(* CODESYS project NTC-Tester-Techmicron.project
   Version: 0.0.0.0
   Title: NTC-Tester-Techmicron
   Author: ekoru

Project tree, tasks and I/O mapping:
  MyController : TM241CE40R, Schneider Electric, order no. TM241CE40R, version 5.0.8.2
    application Application
      libraries: Network, 3.5.7.0 (3S - Smart Software Solutions GmbH)
      task MAST (cyclic, interval 20 ms, priority 15, watchdog 100 ms x 1) calls Input, Output, Auto_Sequence, Man_Sequence, DMM_Connection, Test_Result
      global variables GVL
      program Input [LD]
      program Output [LD]
      program Auto_Sequence [LD]
      program Man_Sequence [LD]
      program DMM_Connection [LD]
      program Test_Result [LD]
    DI : Digital Inputs, Schneider Electric, version 5.0.8.2
        input  idwDI_IDW0 : DWORD  // IDW0
        input  ibDI_IB1 : BYTE  // IB1
    DQ : Digital Outputs, Schneider Electric, version 5.0.8.2
        output qwDQ_QW0 : WORD  // QW0
        output qbDQ_QB1 : BYTE  // QB1
    Counters : Counters, Schneider Electric, version 5.0.8.2
    Pulse_Generators : Pulse Generators, Schneider Electric, version 5.0.8.2
    Cartridge_1 : Cartridge, Schneider Electric, version 5.0.8.2
    Cartridge_2 : Cartridge, Schneider Electric, version 5.0.8.2
    IO_Bus : IO bus - TM3, Schneider Electric, version 5.0.8.2
    COM_Bus : COM bus, Schneider Electric, version 5.0.8.2
    Ethernet_1 : Ethernet Network, Schneider Electric, version 5.0.8.2
        settings: IPAddress = [192, 168, 1, 10]; SubnetMask = [255, 255, 255, 0]; WebServer = TRUE; FTP Server = FALSE; SoMachine Protocol = TRUE; Modbus Server = FALSE; NetManage Protocol = TRUE; SNMP protocol = FALSE; Enable Routing = FALSE; WebVisu protocol = FALSE; DHCP Server Active = TRUE
    Serial_Line_1 : Serial line, Schneider Electric, version 5.0.8.2
      Machine_Expert_Network_Manager : Machine Expert-Network Manager, Schneider Electric, version 4.0.0.3
    Serial_Line_2 : Serial line, Schneider Electric, version 5.0.8.2
      Modbus_Manager : Modbus Manager, Schneider Electric, version 4.0.0.3
*)

// MyController/Application/GVL
{attribute 'qualified_only'}
VAR_GLOBAL
	// Input
	// S1
	Cyl_A_min AT %IX0.1: BOOL;
	// S2
	Cyl_A_max AT %IX0.0: BOOL;
	// S3
	Cyl_B_min AT %IX0.2: BOOL;
	// S4
	Cyl_B_max AT %IX0.3: BOOL;
	// S5
	Jig_Sensor AT %IX0.4: BOOL;
	// S6
	Sw_EMG AT %IX0.8: BOOL;
	// S7
	Sw_Auto AT %IX0.9: BOOL;
	// S8
	Sw_PB_Left AT %IX0.10: BOOL;
	// S9
	Sw_PB_Right AT %IX0.11: BOOL;
	// Timer Cyl A min
	Timer_Cyl_A_min: BOOL;
	Timer_Cyl_A_max: BOOL;
	Timer_Cyl_B_min: BOOL;
	Timer_Cyl_B_max: BOOL;
	Timer_Jig_Sensor: BOOL;
	Trigger_Cycle: BOOL;
	
	// Output
	Led_Red_1 AT %QX0.0: BOOL;
	Led_Red_2 AT %QX0.1: BOOL;
	Led_Red_3 AT %QX0.2: BOOL;
	Led_Red_4 AT %QX0.3: BOOL;
	Led_Green_1 AT %QX0.4: BOOL;
	Led_Green_2 AT %QX0.5: BOOL;
	Led_Green_3 AT %QX0.6: BOOL;
	Led_Green_4 AT %QX0.7: BOOL;
	Sol_Cyl_A AT %QX0.8: BOOL;
	Sol_Cyl_B AT %QX0.9: BOOL;
	Buzzer AT %QX0.10: BOOL;
	Coil_K1 AT %QX0.11: BOOL;
	Coil_K2 AT %QX0.12: BOOL;
	Coil_K3 AT %QX0.13: BOOL;
	Coil_K4 AT %QX0.14: BOOL;
	
	// Sequence
	Seq_Cyl_A_Forward: BOOL;
	Seq_Cyl_B_Down: BOOL;
	Seq_Test_1: BOOL;
	Seq_Test_2: BOOL;
	Seq_Test_3: BOOL;
	Seq_Test_4: BOOL;
	Seq_Cyl_B_Up: BOOL;
	Seq_Cyl_A_Backward: BOOL;
	Seq_Done: BOOL;
	Sw_PB_Right_Cycle: BOOL;
	Man_Done: BOOL;
	Man_Cyl_A_Forward: BOOL;
	Man_Cyl_B_Down: BOOL;
	Man_Test_1: BOOL;
	Man_Test_2: BOOL;
	Man_Test_3: BOOL;
	Man_Test_4: BOOL;
	Man_Cyl_B_Up: BOOL;
	Man_Cyl_A_Backward: BOOL;
	Sw_EMG_Cycle: BOOL;
	TCP_Connected: BOOL;
	DMM_Connected: BOOL;
	Test_1_Write: BOOL;
	Test_1_Read: BOOL;
	
	Man_Test_1_Write: BOOL;
	Man_Test_1_Read: BOOL;
	Man_Test_2_Write: BOOL;
	Man_Test_2_Read: BOOL;
	Man_Test_3_Write: BOOL;
	Man_Test_3_Read: BOOL;
	Man_Test_4_Write: BOOL;
	Man_Test_4_Read: BOOL;
	Seq_Test_1_Write: BOOL;
	Seq_Test_1_Read: BOOL;
	Seq_Test_2_Write: BOOL;
	Seq_Test_2_Read: BOOL;
	Seq_Test_3_Write: BOOL;
	Seq_Test_3_Read: BOOL;
	Seq_Test_4_Write: BOOL;
	Seq_Test_4_Read: BOOL;
	
	Res_Value: REAL;
	Spec_Min_Value: REAL:= 7000;
	Spec_Max_Value: REAL:= 9000;
	
	Seq_Test_1_Done: BOOL;
	Seq_Test_2_Done: BOOL;
	Seq_Test_3_Done: BOOL;
	Seq_Test_4_Done: BOOL;
	Man_Test_1_Done: BOOL;
	Man_Test_2_Done: BOOL;
	Man_Test_3_Done: BOOL;
	Man_Test_4_Done: BOOL;
END_VAR

// MyController/Application/Input
PROGRAM Input
VAR
	T_Cyl_A_min: TON;
	T_Cyl_A_max: TON;
	T_Cyl_B_min: TON;
	T_Cyl_B_max: TON;
	T_Cyl_Jig_Sensor: TON;
	T_Sw_PB_Left: TON;
	T_Sw_PB_Left_Out: BOOL;
	T_Sw_PB_Right: TON;
	T_Sw_PB_Right_Out: BOOL;
END_VAR
VAR // added by the converter: edge detectors and wires of the graphical bodies
    _rt1, _rt2 : R_TRIG;
    _ft1 : F_TRIG;
END_VAR

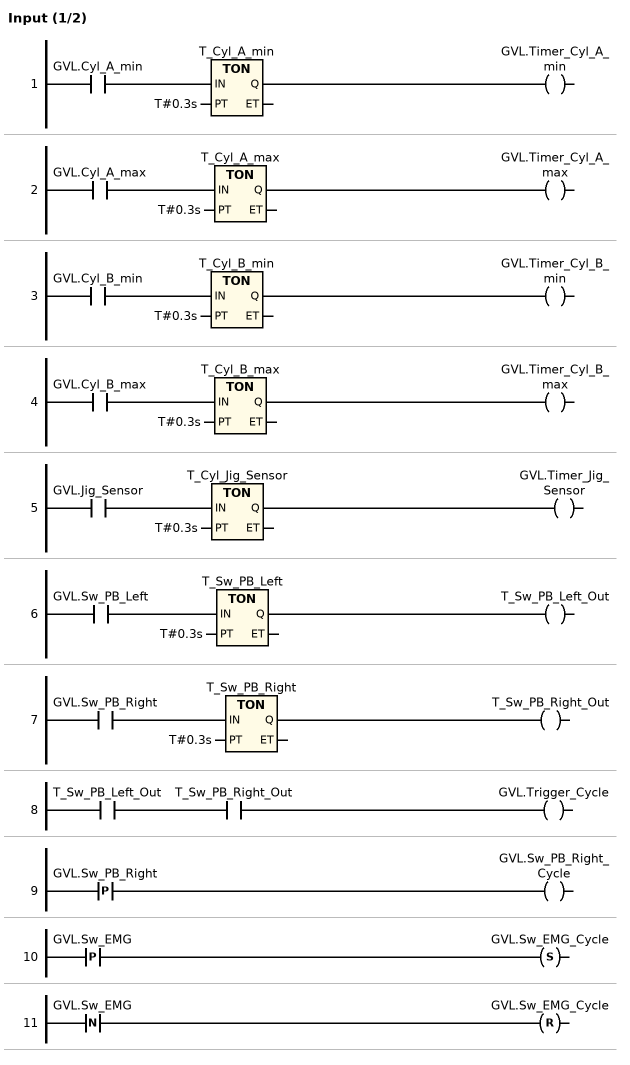
// NETWORK 1
T_Cyl_A_min(IN := GVL.Cyl_A_min, PT := T#0.3s); // TON
GVL.Timer_Cyl_A_min := T_Cyl_A_min.Q;

// NETWORK 2
T_Cyl_A_max(IN := GVL.Cyl_A_max, PT := T#0.3s); // TON
GVL.Timer_Cyl_A_max := T_Cyl_A_max.Q;

// NETWORK 3
T_Cyl_B_min(IN := GVL.Cyl_B_min, PT := T#0.3s); // TON
GVL.Timer_Cyl_B_min := T_Cyl_B_min.Q;

// NETWORK 4
T_Cyl_B_max(IN := GVL.Cyl_B_max, PT := T#0.3s); // TON
GVL.Timer_Cyl_B_max := T_Cyl_B_max.Q;

// NETWORK 5
T_Cyl_Jig_Sensor(IN := GVL.Jig_Sensor, PT := T#0.3s); // TON
GVL.Timer_Jig_Sensor := T_Cyl_Jig_Sensor.Q;

// NETWORK 6
T_Sw_PB_Left(IN := GVL.Sw_PB_Left, PT := T#0.3s); // TON
T_Sw_PB_Left_Out := T_Sw_PB_Left.Q;

// NETWORK 7
T_Sw_PB_Right(IN := GVL.Sw_PB_Right, PT := T#0.3s); // TON
T_Sw_PB_Right_Out := T_Sw_PB_Right.Q;

// NETWORK 8
GVL.Trigger_Cycle := T_Sw_PB_Left_Out AND T_Sw_PB_Right_Out;

// NETWORK 9
_rt1(CLK := GVL.Sw_PB_Right);
GVL.Sw_PB_Right_Cycle := _rt1.Q;

// NETWORK 10
_rt2(CLK := GVL.Sw_EMG);
GVL.Sw_EMG_Cycle S= _rt2.Q;

// NETWORK 11
_ft1(CLK := GVL.Sw_EMG);
GVL.Sw_EMG_Cycle R= _ft1.Q;

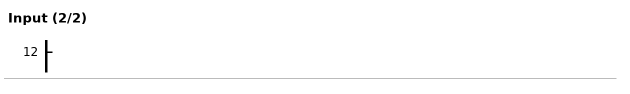
// NETWORK 12

END_PROGRAM

// MyController/Application/Output
PROGRAM Output
VAR	
END_VAR

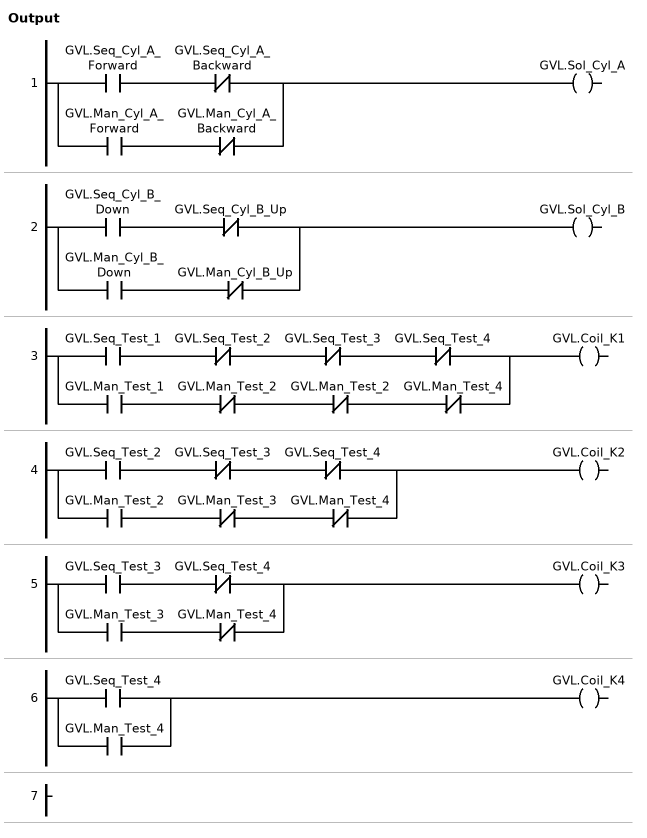
// NETWORK 1
GVL.Sol_Cyl_A := GVL.Seq_Cyl_A_Forward AND NOT GVL.Seq_Cyl_A_Backward OR GVL.Man_Cyl_A_Forward AND NOT GVL.Man_Cyl_A_Backward;

// NETWORK 2
GVL.Sol_Cyl_B := GVL.Seq_Cyl_B_Down AND NOT GVL.Seq_Cyl_B_Up OR GVL.Man_Cyl_B_Down AND NOT GVL.Man_Cyl_B_Up;

// NETWORK 3
GVL.Coil_K1 := GVL.Seq_Test_1 AND NOT GVL.Seq_Test_2 AND NOT GVL.Seq_Test_3 AND NOT GVL.Seq_Test_4 OR GVL.Man_Test_1 AND NOT GVL.Man_Test_2 AND NOT GVL.Man_Test_2 AND NOT GVL.Man_Test_4;

// NETWORK 4
GVL.Coil_K2 := GVL.Seq_Test_2 AND NOT GVL.Seq_Test_3 AND NOT GVL.Seq_Test_4 OR GVL.Man_Test_2 AND NOT GVL.Man_Test_3 AND NOT GVL.Man_Test_4;

// NETWORK 5
GVL.Coil_K3 := GVL.Seq_Test_3 AND NOT GVL.Seq_Test_4 OR GVL.Man_Test_3 AND NOT GVL.Man_Test_4;

// NETWORK 6
GVL.Coil_K4 := GVL.Seq_Test_4 OR GVL.Man_Test_4;

// NETWORK 7

END_PROGRAM

// MyController/Application/Auto_Sequence
PROGRAM Auto_Sequence
VAR
	Init_State: BOOL;
	T_Seq_Test_1: TON;
	Test_1_Done: BOOL;
	T_Seq_Test_2: TON;
	Test_2_Done: BOOL;
	T_Seq_Test_3: TON;
	Test_3_Done: BOOL;
	T_Seq_Test_4: TON;
	Test_4_Done: BOOL;
	T_Seq_Test_1_Contact: TON;
	T_Seq_Test_1_Write: TON;
	T_Seq_Test_2_Contact: TON;
	T_Seq_Test_2_Write: TON;
	T_Seq_Test_3_Contact: TON;
	T_Seq_Test_3_Write: TON;
	T_Seq_Test_4_Contact: TON;
	T_Seq_Test_4_Write: TON;
END_VAR
VAR // added by the converter: edge detectors and wires of the graphical bodies
    _ft1 : F_TRIG;
END_VAR

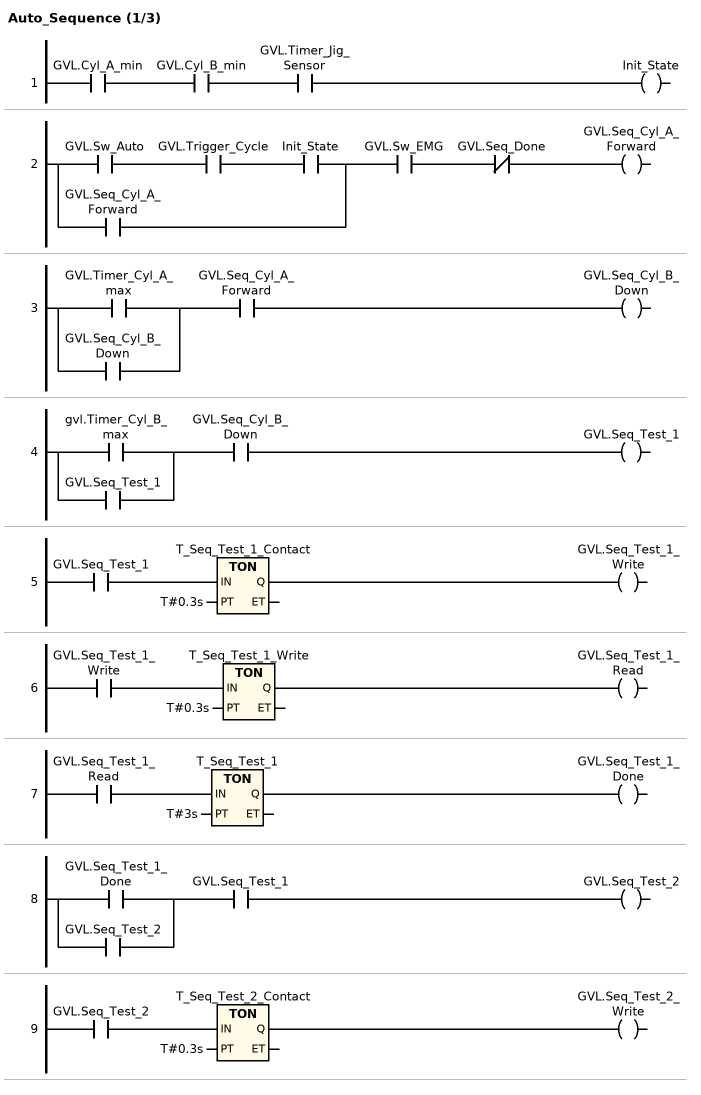
// NETWORK 1
Init_State := GVL.Cyl_A_min AND GVL.Cyl_B_min AND GVL.Timer_Jig_Sensor;

// NETWORK 2
GVL.Seq_Cyl_A_Forward := (GVL.Sw_Auto AND GVL.Trigger_Cycle AND Init_State OR GVL.Seq_Cyl_A_Forward) AND GVL.Sw_EMG AND NOT GVL.Seq_Done;

// NETWORK 3
GVL.Seq_Cyl_B_Down := (GVL.Timer_Cyl_A_max OR GVL.Seq_Cyl_B_Down) AND GVL.Seq_Cyl_A_Forward;

// NETWORK 4
GVL.Seq_Test_1 := (gvl.Timer_Cyl_B_max OR GVL.Seq_Test_1) AND GVL.Seq_Cyl_B_Down;

// NETWORK 5
T_Seq_Test_1_Contact(IN := GVL.Seq_Test_1, PT := T#0.3s); // TON
GVL.Seq_Test_1_Write := T_Seq_Test_1_Contact.Q;

// NETWORK 6
T_Seq_Test_1_Write(IN := GVL.Seq_Test_1_Write, PT := T#0.3s); // TON
GVL.Seq_Test_1_Read := T_Seq_Test_1_Write.Q;

// NETWORK 7
T_Seq_Test_1(IN := GVL.Seq_Test_1_Read, PT := T#3s); // TON
GVL.Seq_Test_1_Done := T_Seq_Test_1.Q;

// NETWORK 8
GVL.Seq_Test_2 := (GVL.Seq_Test_1_Done OR GVL.Seq_Test_2) AND GVL.Seq_Test_1;

// NETWORK 9
T_Seq_Test_2_Contact(IN := GVL.Seq_Test_2, PT := T#0.3s); // TON
GVL.Seq_Test_2_Write := T_Seq_Test_2_Contact.Q;

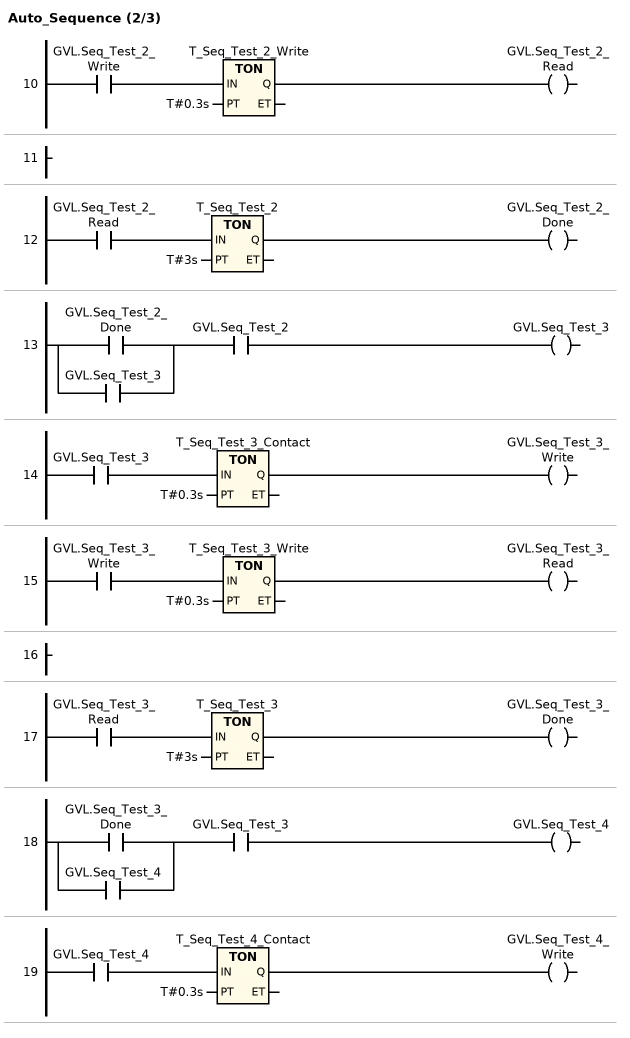
// NETWORK 10
T_Seq_Test_2_Write(IN := GVL.Seq_Test_2_Write, PT := T#0.3s); // TON
GVL.Seq_Test_2_Read := T_Seq_Test_2_Write.Q;

// NETWORK 11

// NETWORK 12
T_Seq_Test_2(IN := GVL.Seq_Test_2_Read, PT := T#3s); // TON
GVL.Seq_Test_2_Done := T_Seq_Test_2.Q;

// NETWORK 13
GVL.Seq_Test_3 := (GVL.Seq_Test_2_Done OR GVL.Seq_Test_3) AND GVL.Seq_Test_2;

// NETWORK 14
T_Seq_Test_3_Contact(IN := GVL.Seq_Test_3, PT := T#0.3s); // TON
GVL.Seq_Test_3_Write := T_Seq_Test_3_Contact.Q;

// NETWORK 15
T_Seq_Test_3_Write(IN := GVL.Seq_Test_3_Write, PT := T#0.3s); // TON
GVL.Seq_Test_3_Read := T_Seq_Test_3_Write.Q;

// NETWORK 16

// NETWORK 17
T_Seq_Test_3(IN := GVL.Seq_Test_3_Read, PT := T#3s); // TON
GVL.Seq_Test_3_Done := T_Seq_Test_3.Q;

// NETWORK 18
GVL.Seq_Test_4 := (GVL.Seq_Test_3_Done OR GVL.Seq_Test_4) AND GVL.Seq_Test_3;

// NETWORK 19
T_Seq_Test_4_Contact(IN := GVL.Seq_Test_4, PT := T#0.3s); // TON
GVL.Seq_Test_4_Write := T_Seq_Test_4_Contact.Q;

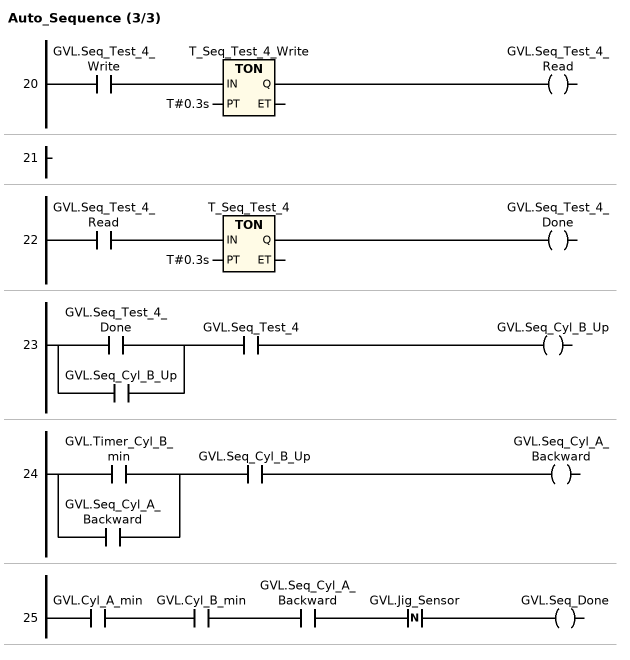
// NETWORK 20
T_Seq_Test_4_Write(IN := GVL.Seq_Test_4_Write, PT := T#0.3s); // TON
GVL.Seq_Test_4_Read := T_Seq_Test_4_Write.Q;

// NETWORK 21

// NETWORK 22
T_Seq_Test_4(IN := GVL.Seq_Test_4_Read, PT := T#0.3s); // TON
GVL.Seq_Test_4_Done := T_Seq_Test_4.Q;

// NETWORK 23
GVL.Seq_Cyl_B_Up := (GVL.Seq_Test_4_Done OR GVL.Seq_Cyl_B_Up) AND GVL.Seq_Test_4;

// NETWORK 24
GVL.Seq_Cyl_A_Backward := (GVL.Timer_Cyl_B_min OR GVL.Seq_Cyl_A_Backward) AND GVL.Seq_Cyl_B_Up;

// NETWORK 25
_ft1(CLK := GVL.Jig_Sensor);
GVL.Seq_Done := GVL.Cyl_A_min AND GVL.Cyl_B_min AND GVL.Seq_Cyl_A_Backward AND _ft1.Q;

END_PROGRAM

// MyController/Application/Man_Sequence
PROGRAM Man_Sequence
VAR
	Init_State: BOOL;
	Test_1_Done: BOOL;
	Test_2_Done: BOOL;
	Test_3_Done: BOOL;
	Test_4_Done: BOOL;
	T_Man_Test_1_Contact: TON;
	T_Man_Test_1_Write: TON;
	T_Man_Test_1_Read: TON;
	T_Man_Test_2_Contact: TON;
	T_Man_Test_2_Write: TON;
	T_Man_Test_2_Read: TON;
	T_Man_Test_3_Contact: TON;
	T_Man_Test_3_Write: TON;
	T_Man_Test_3_Read: TON;
	T_Man_Test_4_Contact: TON;
	T_Man_Test_4_Write: TON;
	T_Man_Test_4_Read: TON;
END_VAR

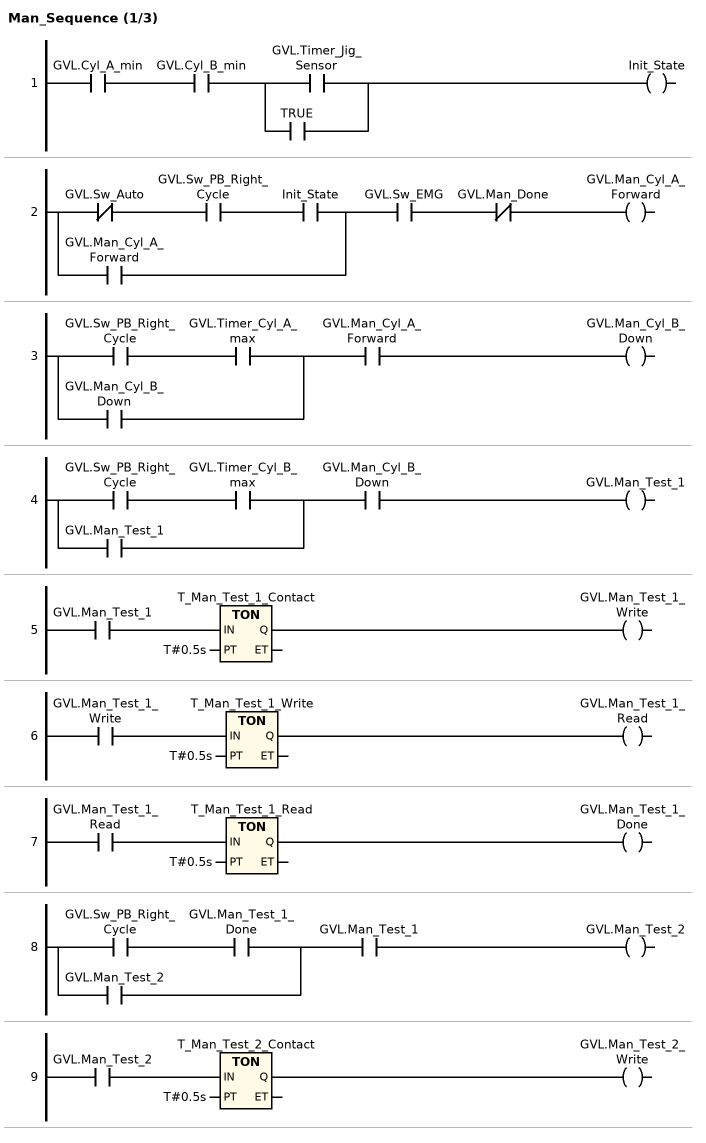
// NETWORK 1
Init_State := GVL.Cyl_A_min AND GVL.Cyl_B_min AND (GVL.Timer_Jig_Sensor OR TRUE);

// NETWORK 2
GVL.Man_Cyl_A_Forward := (NOT GVL.Sw_Auto AND GVL.Sw_PB_Right_Cycle AND Init_State OR GVL.Man_Cyl_A_Forward) AND GVL.Sw_EMG AND NOT GVL.Man_Done;

// NETWORK 3
GVL.Man_Cyl_B_Down := (GVL.Sw_PB_Right_Cycle AND GVL.Timer_Cyl_A_max OR GVL.Man_Cyl_B_Down) AND GVL.Man_Cyl_A_Forward;

// NETWORK 4
GVL.Man_Test_1 := (GVL.Sw_PB_Right_Cycle AND GVL.Timer_Cyl_B_max OR GVL.Man_Test_1) AND GVL.Man_Cyl_B_Down;

// NETWORK 5
T_Man_Test_1_Contact(IN := GVL.Man_Test_1, PT := T#0.5s); // TON
GVL.Man_Test_1_Write := T_Man_Test_1_Contact.Q;

// NETWORK 6
T_Man_Test_1_Write(IN := GVL.Man_Test_1_Write, PT := T#0.5s); // TON
GVL.Man_Test_1_Read := T_Man_Test_1_Write.Q;

// NETWORK 7
T_Man_Test_1_Read(IN := GVL.Man_Test_1_Read, PT := T#0.5s); // TON
GVL.Man_Test_1_Done := T_Man_Test_1_Read.Q;

// NETWORK 8
GVL.Man_Test_2 := (GVL.Sw_PB_Right_Cycle AND GVL.Man_Test_1_Done OR GVL.Man_Test_2) AND GVL.Man_Test_1;

// NETWORK 9
T_Man_Test_2_Contact(IN := GVL.Man_Test_2, PT := T#0.5s); // TON
GVL.Man_Test_2_Write := T_Man_Test_2_Contact.Q;

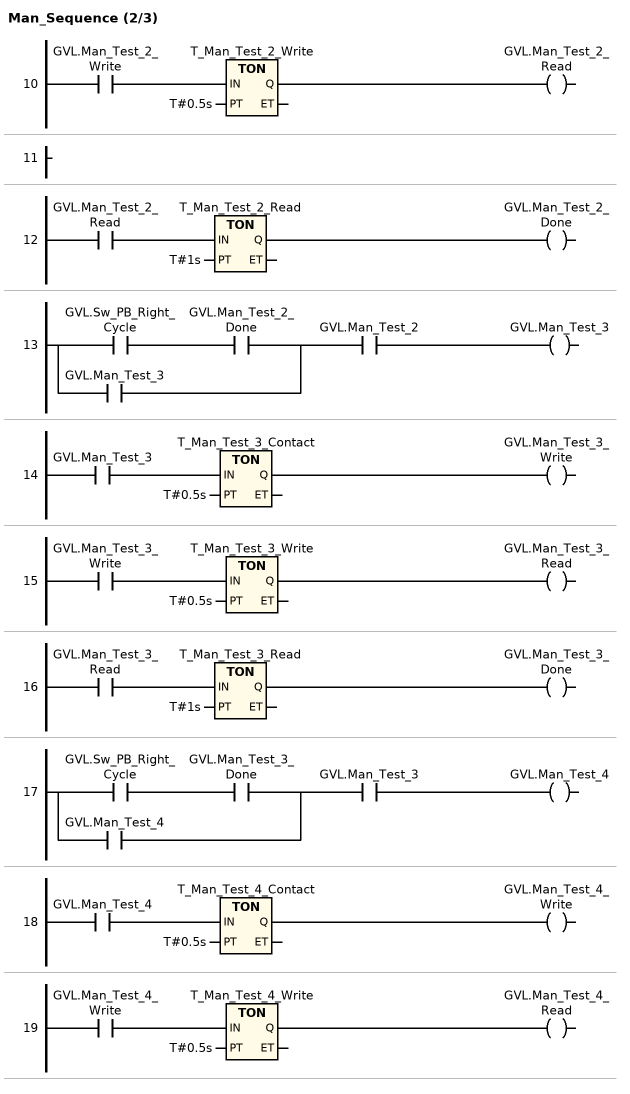
// NETWORK 10
T_Man_Test_2_Write(IN := GVL.Man_Test_2_Write, PT := T#0.5s); // TON
GVL.Man_Test_2_Read := T_Man_Test_2_Write.Q;

// NETWORK 11

// NETWORK 12
T_Man_Test_2_Read(IN := GVL.Man_Test_2_Read, PT := T#1s); // TON
GVL.Man_Test_2_Done := T_Man_Test_2_Read.Q;

// NETWORK 13
GVL.Man_Test_3 := (GVL.Sw_PB_Right_Cycle AND GVL.Man_Test_2_Done OR GVL.Man_Test_3) AND GVL.Man_Test_2;

// NETWORK 14
T_Man_Test_3_Contact(IN := GVL.Man_Test_3, PT := T#0.5s); // TON
GVL.Man_Test_3_Write := T_Man_Test_3_Contact.Q;

// NETWORK 15
T_Man_Test_3_Write(IN := GVL.Man_Test_3_Write, PT := T#0.5s); // TON
GVL.Man_Test_3_Read := T_Man_Test_3_Write.Q;

// NETWORK 16
T_Man_Test_3_Read(IN := GVL.Man_Test_3_Read, PT := T#1s); // TON
GVL.Man_Test_3_Done := T_Man_Test_3_Read.Q;

// NETWORK 17
GVL.Man_Test_4 := (GVL.Sw_PB_Right_Cycle AND GVL.Man_Test_3_Done OR GVL.Man_Test_4) AND GVL.Man_Test_3;

// NETWORK 18
T_Man_Test_4_Contact(IN := GVL.Man_Test_4, PT := T#0.5s); // TON
GVL.Man_Test_4_Write := T_Man_Test_4_Contact.Q;

// NETWORK 19
T_Man_Test_4_Write(IN := GVL.Man_Test_4_Write, PT := T#0.5s); // TON
GVL.Man_Test_4_Read := T_Man_Test_4_Write.Q;

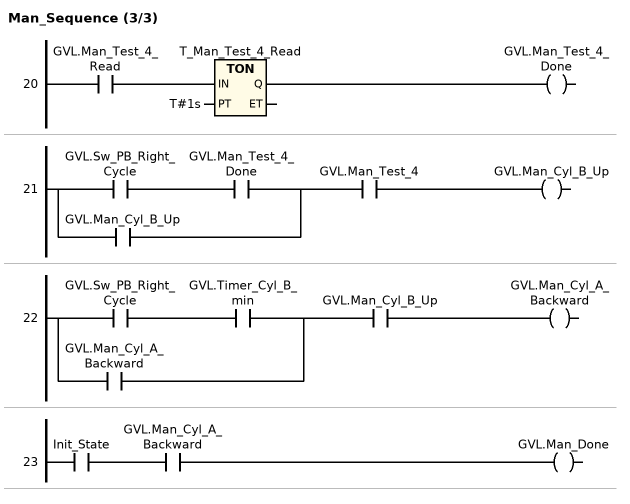
// NETWORK 20
T_Man_Test_4_Read(IN := GVL.Man_Test_4_Read, PT := T#1s); // TON
GVL.Man_Test_4_Done := T_Man_Test_4_Read.Q;

// NETWORK 21
GVL.Man_Cyl_B_Up := (GVL.Sw_PB_Right_Cycle AND GVL.Man_Test_4_Done OR GVL.Man_Cyl_B_Up) AND GVL.Man_Test_4;

// NETWORK 22
GVL.Man_Cyl_A_Backward := (GVL.Sw_PB_Right_Cycle AND GVL.Timer_Cyl_B_min OR GVL.Man_Cyl_A_Backward) AND GVL.Man_Cyl_B_Up;

// NETWORK 23
GVL.Man_Done := Init_State AND GVL.Man_Cyl_A_Backward;

END_PROGRAM

// MyController/Application/DMM_Connection
PROGRAM DMM_Connection
VAR
	TCP_Client_0: NBS.TCP_Client;
	IP_Address: NBS.IP_ADDR;
	Connect: BOOL;
	Connected: BOOL;
	TCP_Write_0: NBS.TCP_Write;
	hConnection_0: CAA.HANDLE;
	Write: BOOL;
	//DataSend: STRING := 'MEAS?$L';
	DataSend: STRING := 'MEAS:FRES?$L';
	//DataSend: STRING := ':CALC:FRES:LIM<1>:FAIL?$L';
	DataReceived: STRING(255);
	Data_Sent: BOOL;
	Set_String: BOOL;
	TCP_Read_0: NBS.TCP_Read;
	Read: BOOL;
	TCP_WriteBuffer_0: NBS.TCP_WriteBuffer;
	Send_Buffer: CAA.HANDLE;
	Data_Received: BOOL;
	TP_0: TP;
	TP_1: TP;
	Man_Read_1: BOOL;
	TP_Man_Read_1: TP;
	TP_Man_Read_2: TP;
	Man_Read_2: BOOL;
	TP_Man_Read_3: TP;
	Man_Read_3: BOOL;
	Man_Read_4: BOOL;
	TP_Man_Read_4: TP;
	TP_Seq_Read_1: TP;
	Seq_Read_1: BOOL;
	TP_Seq_Read_2: TP;
	Seq_Read_2: BOOL;
	TP_Seq_Read_3: TP;
	Seq_Read_3: BOOL;
	TP_Seq_Read_4: TP;
	Seq_Read_4: BOOL;
	Man_Write_1: BOOL;
	TP_Man_Write_1: TP;
	TP_Man_Write_2: TP;
	Man_Write_2: BOOL;
	TP_Man_Write_3: TP;
	Man_Write_3: BOOL;
	TP_Man_Write_4: TP;
	Man_Write_4: BOOL;
	TP_Seq_Write_1: TP;
	Seq_Write_1: BOOL;
	TP_Seq_Write_2: TP;
	Seq_Write_2: BOOL;
	TP_Seq_Write_3: TP;
	Seq_Write_3: BOOL;
	TP_Seq_Write_4: TP;
	Seq_Write_4: BOOL;
END_VAR
VAR // added by the converter: edge detectors and wires of the graphical bodies
    _rt1 : R_TRIG;
END_VAR

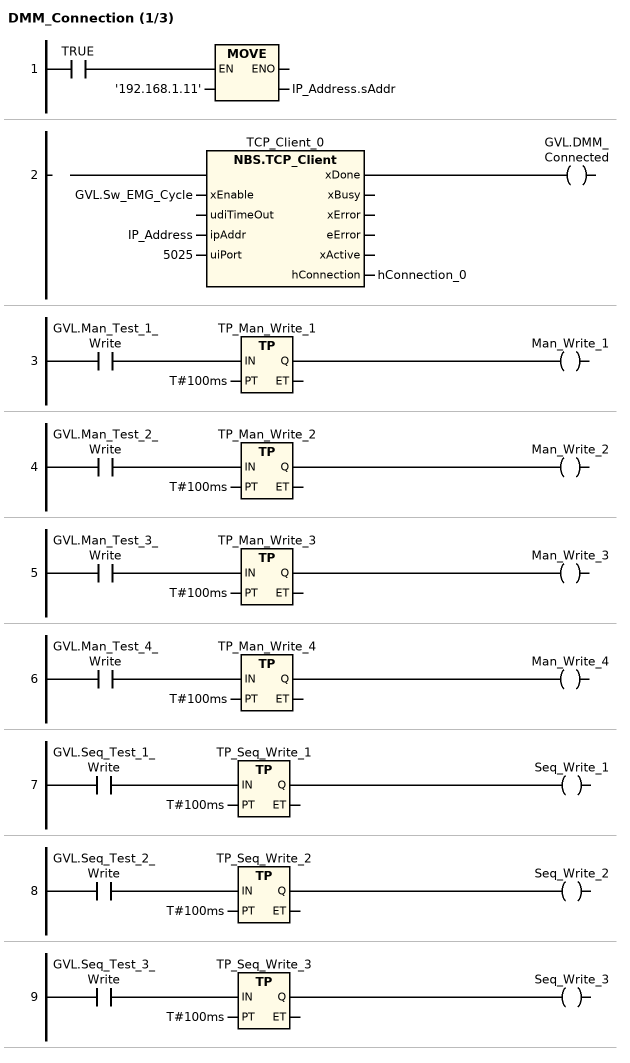
// NETWORK 1
IP_Address.sAddr := '192.168.1.11';

// NETWORK 2
TCP_Client_0(xEnable := GVL.Sw_EMG_Cycle, ipAddr := IP_Address, uiPort := 5025, hConnection => hConnection_0); // NBS.TCP_Client
GVL.DMM_Connected := TCP_Client_0.xDone;

// NETWORK 3
TP_Man_Write_1(IN := GVL.Man_Test_1_Write, PT := T#100ms); // TP
Man_Write_1 := TP_Man_Write_1.Q;

// NETWORK 4
TP_Man_Write_2(IN := GVL.Man_Test_2_Write, PT := T#100ms); // TP
Man_Write_2 := TP_Man_Write_2.Q;

// NETWORK 5
TP_Man_Write_3(IN := GVL.Man_Test_3_Write, PT := T#100ms); // TP
Man_Write_3 := TP_Man_Write_3.Q;

// NETWORK 6
TP_Man_Write_4(IN := GVL.Man_Test_4_Write, PT := T#100ms); // TP
Man_Write_4 := TP_Man_Write_4.Q;

// NETWORK 7
TP_Seq_Write_1(IN := GVL.Seq_Test_1_Write, PT := T#100ms); // TP
Seq_Write_1 := TP_Seq_Write_1.Q;

// NETWORK 8
TP_Seq_Write_2(IN := GVL.Seq_Test_2_Write, PT := T#100ms); // TP
Seq_Write_2 := TP_Seq_Write_2.Q;

// NETWORK 9
TP_Seq_Write_3(IN := GVL.Seq_Test_3_Write, PT := T#100ms); // TP
Seq_Write_3 := TP_Seq_Write_3.Q;

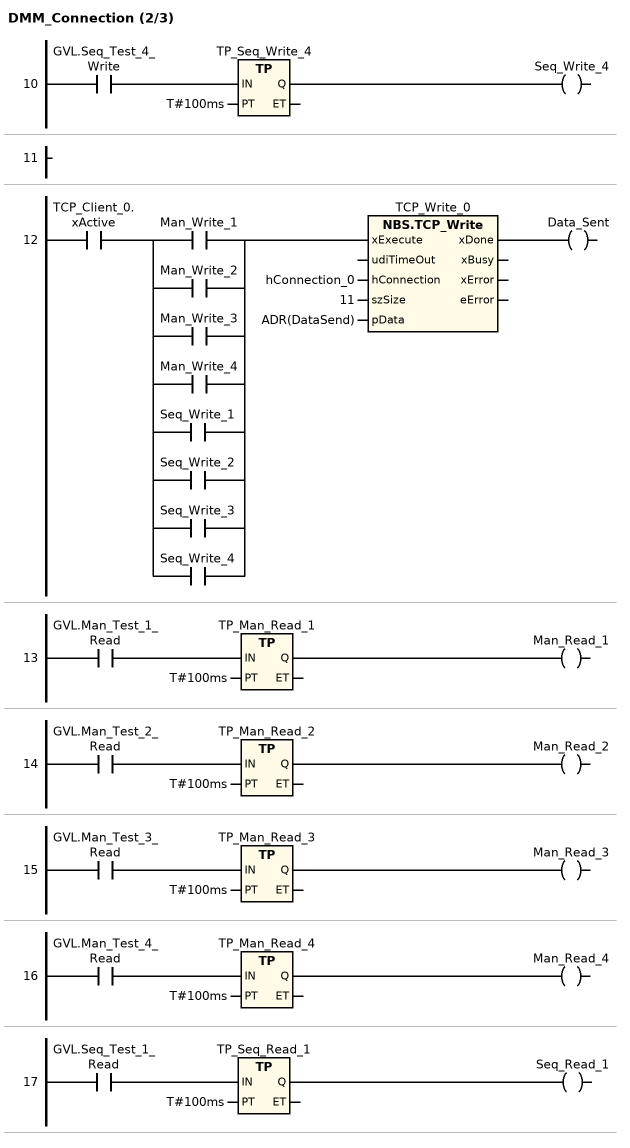
// NETWORK 10
TP_Seq_Write_4(IN := GVL.Seq_Test_4_Write, PT := T#100ms); // TP
Seq_Write_4 := TP_Seq_Write_4.Q;

// NETWORK 11

// NETWORK 12
TCP_Write_0(
    xExecute := TCP_Client_0.xActive AND (Man_Write_1 OR Man_Write_2 OR Man_Write_3 OR Man_Write_4 OR Seq_Write_1 OR Seq_Write_2 OR Seq_Write_3 OR Seq_Write_4),
    hConnection := hConnection_0,
    szSize := 11,
    pData := ADR(DataSend)); // NBS.TCP_Write
Data_Sent := TCP_Write_0.xDone;

// NETWORK 13
TP_Man_Read_1(IN := GVL.Man_Test_1_Read, PT := T#100ms); // TP
Man_Read_1 := TP_Man_Read_1.Q;

// NETWORK 14
TP_Man_Read_2(IN := GVL.Man_Test_2_Read, PT := T#100ms); // TP
Man_Read_2 := TP_Man_Read_2.Q;

// NETWORK 15
TP_Man_Read_3(IN := GVL.Man_Test_3_Read, PT := T#100ms); // TP
Man_Read_3 := TP_Man_Read_3.Q;

// NETWORK 16
TP_Man_Read_4(IN := GVL.Man_Test_4_Read, PT := T#100ms); // TP
Man_Read_4 := TP_Man_Read_4.Q;

// NETWORK 17
TP_Seq_Read_1(IN := GVL.Seq_Test_1_Read, PT := T#100ms); // TP
Seq_Read_1 := TP_Seq_Read_1.Q;

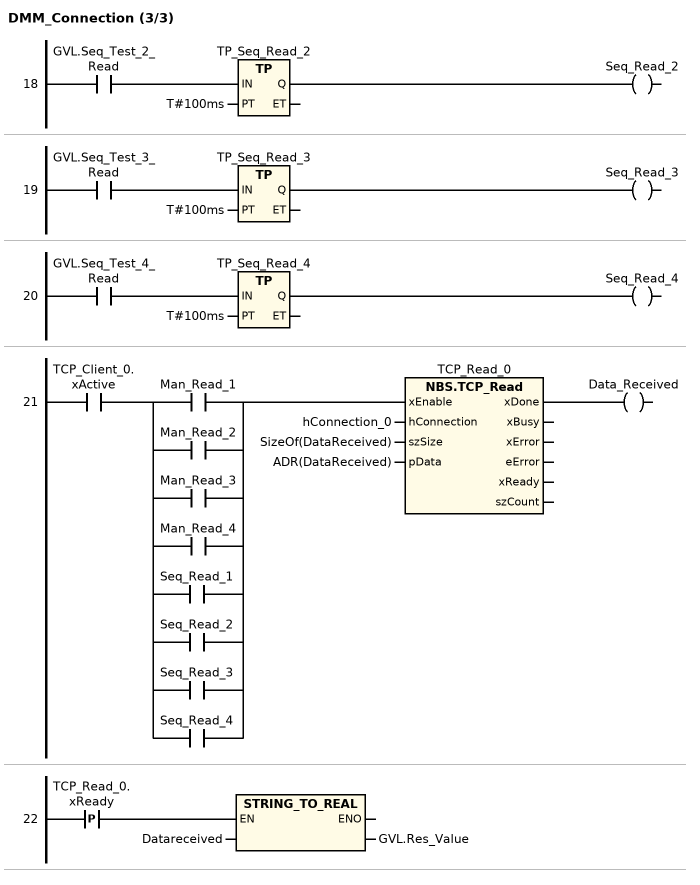
// NETWORK 18
TP_Seq_Read_2(IN := GVL.Seq_Test_2_Read, PT := T#100ms); // TP
Seq_Read_2 := TP_Seq_Read_2.Q;

// NETWORK 19
TP_Seq_Read_3(IN := GVL.Seq_Test_3_Read, PT := T#100ms); // TP
Seq_Read_3 := TP_Seq_Read_3.Q;

// NETWORK 20
TP_Seq_Read_4(IN := GVL.Seq_Test_4_Read, PT := T#100ms); // TP
Seq_Read_4 := TP_Seq_Read_4.Q;

// NETWORK 21
TCP_Read_0(
    xEnable := TCP_Client_0.xActive AND (Man_Read_1 OR Man_Read_2 OR Man_Read_3 OR Man_Read_4 OR Seq_Read_1 OR Seq_Read_2 OR Seq_Read_3 OR Seq_Read_4),
    hConnection := hConnection_0,
    szSize := SizeOf(DataReceived),
    pData := ADR(DataReceived)); // NBS.TCP_Read
Data_Received := TCP_Read_0.xDone;

// NETWORK 22
_rt1(CLK := TCP_Read_0.xReady);
IF _rt1.Q THEN GVL.Res_Value := STRING_TO_REAL(Datareceived); END_IF

END_PROGRAM

// MyController/Application/Test_Result
PROGRAM Test_Result
VAR
	TP_Test_1: TP;
	TP_Test_2: TP;
	TP_Test_3: TP;
	TP_Test_4: TP;
	TP_Trig_1: TP;
	TP_Trig_2: TP;
	TP_Trig_3: TP;
	TP_Trig_4: TP;
END_VAR

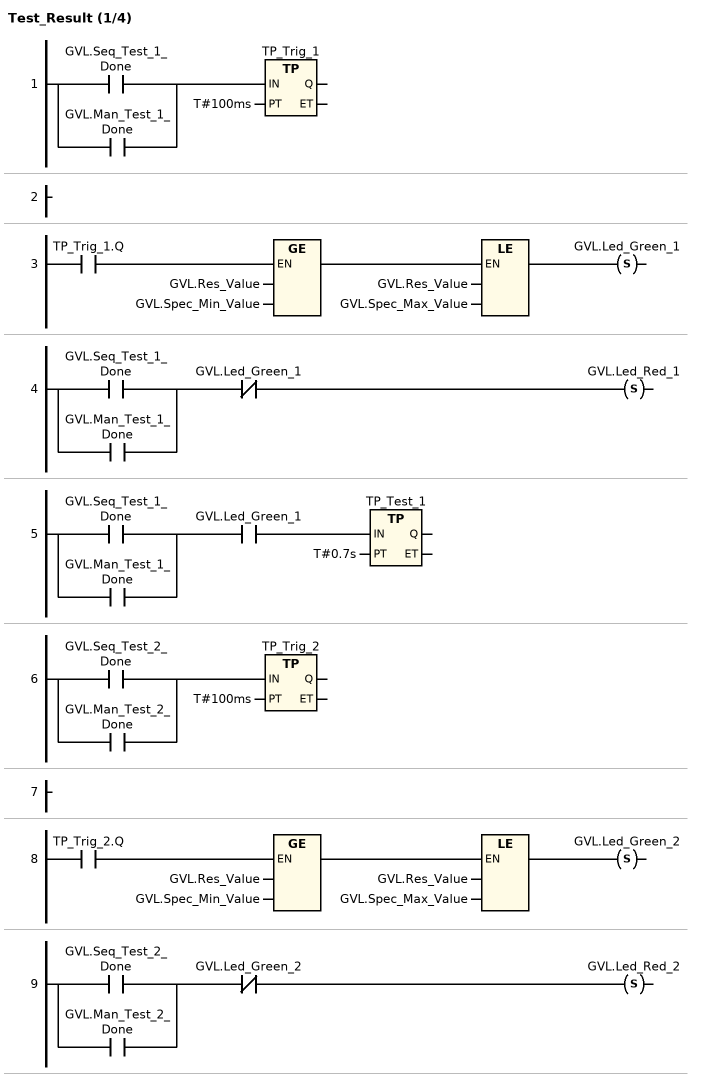
// NETWORK 1
TP_Trig_1(IN := GVL.Seq_Test_1_Done OR GVL.Man_Test_1_Done, PT := T#100ms); // TP

// NETWORK 2

// NETWORK 3
GVL.Led_Green_1 S= TP_Trig_1.Q AND GVL.Res_Value >= GVL.Spec_Min_Value AND GVL.Res_Value <= GVL.Spec_Max_Value;

// NETWORK 4
GVL.Led_Red_1 S= (GVL.Seq_Test_1_Done OR GVL.Man_Test_1_Done) AND NOT GVL.Led_Green_1;

// NETWORK 5
TP_Test_1(IN := (GVL.Seq_Test_1_Done OR GVL.Man_Test_1_Done) AND GVL.Led_Green_1, PT := T#0.7s); // TP

// NETWORK 6
TP_Trig_2(IN := GVL.Seq_Test_2_Done OR GVL.Man_Test_2_Done, PT := T#100ms); // TP

// NETWORK 7

// NETWORK 8
GVL.Led_Green_2 S= TP_Trig_2.Q AND GVL.Res_Value >= GVL.Spec_Min_Value AND GVL.Res_Value <= GVL.Spec_Max_Value;

// NETWORK 9
GVL.Led_Red_2 S= (GVL.Seq_Test_2_Done OR GVL.Man_Test_2_Done) AND NOT GVL.Led_Green_2;

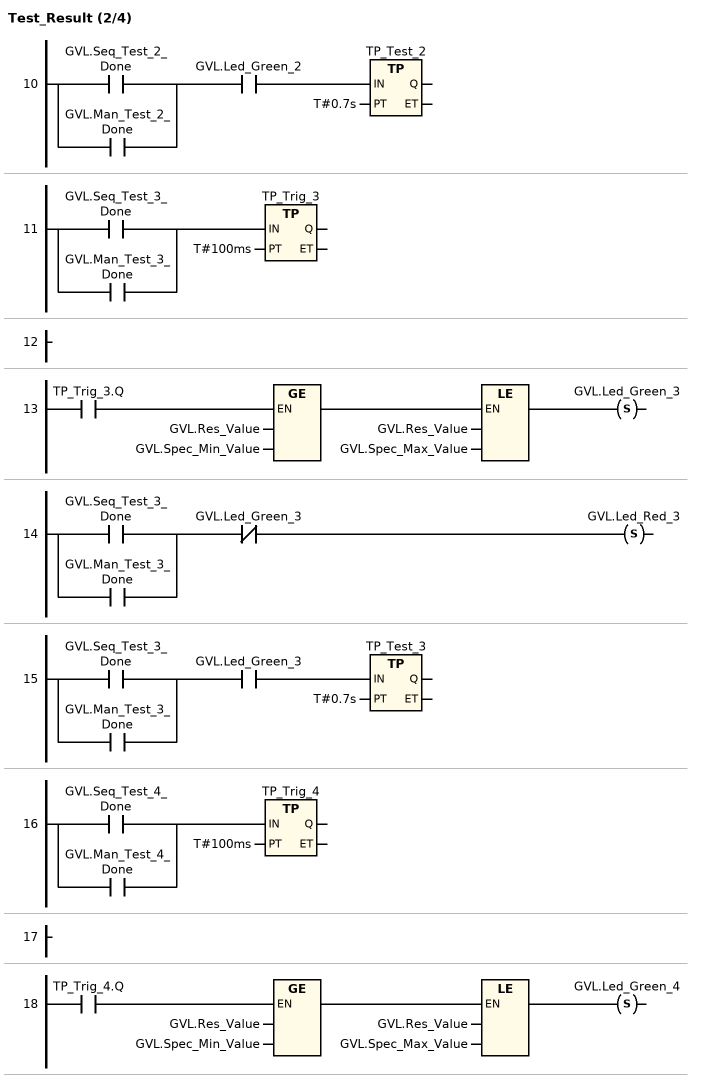
// NETWORK 10
TP_Test_2(IN := (GVL.Seq_Test_2_Done OR GVL.Man_Test_2_Done) AND GVL.Led_Green_2, PT := T#0.7s); // TP

// NETWORK 11
TP_Trig_3(IN := GVL.Seq_Test_3_Done OR GVL.Man_Test_3_Done, PT := T#100ms); // TP

// NETWORK 12

// NETWORK 13
GVL.Led_Green_3 S= TP_Trig_3.Q AND GVL.Res_Value >= GVL.Spec_Min_Value AND GVL.Res_Value <= GVL.Spec_Max_Value;

// NETWORK 14
GVL.Led_Red_3 S= (GVL.Seq_Test_3_Done OR GVL.Man_Test_3_Done) AND NOT GVL.Led_Green_3;

// NETWORK 15
TP_Test_3(IN := (GVL.Seq_Test_3_Done OR GVL.Man_Test_3_Done) AND GVL.Led_Green_3, PT := T#0.7s); // TP

// NETWORK 16
TP_Trig_4(IN := GVL.Seq_Test_4_Done OR GVL.Man_Test_4_Done, PT := T#100ms); // TP

// NETWORK 17

// NETWORK 18
GVL.Led_Green_4 S= TP_Trig_4.Q AND GVL.Res_Value >= GVL.Spec_Min_Value AND GVL.Res_Value <= GVL.Spec_Max_Value;

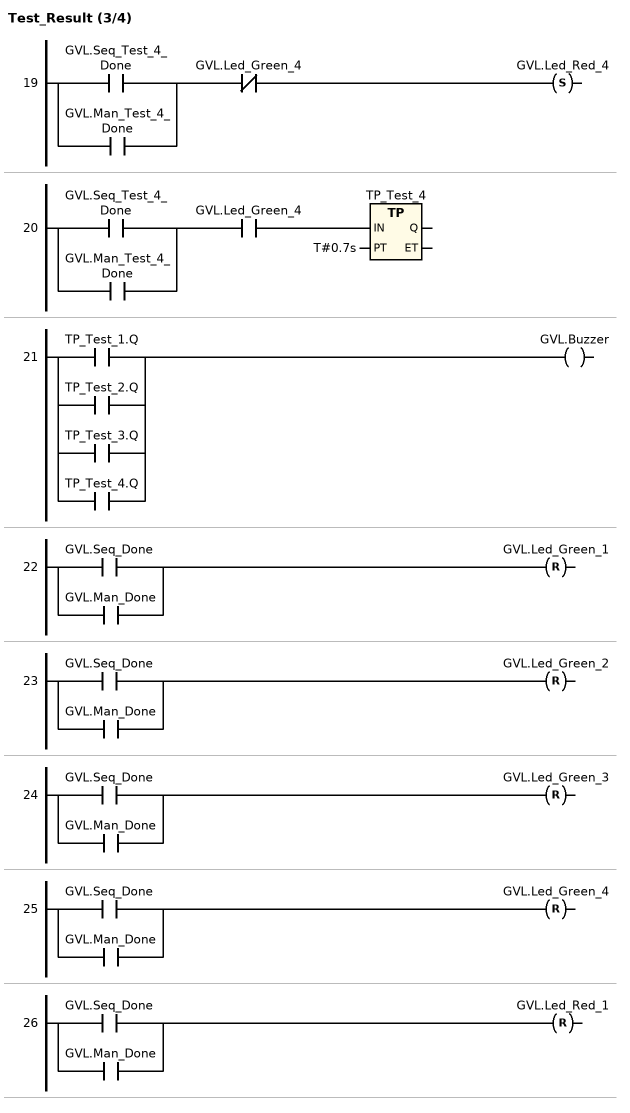
// NETWORK 19
GVL.Led_Red_4 S= (GVL.Seq_Test_4_Done OR GVL.Man_Test_4_Done) AND NOT GVL.Led_Green_4;

// NETWORK 20
TP_Test_4(IN := (GVL.Seq_Test_4_Done OR GVL.Man_Test_4_Done) AND GVL.Led_Green_4, PT := T#0.7s); // TP

// NETWORK 21
GVL.Buzzer := TP_Test_1.Q OR TP_Test_2.Q OR TP_Test_3.Q OR TP_Test_4.Q;

// NETWORK 22
GVL.Led_Green_1 R= GVL.Seq_Done OR GVL.Man_Done;

// NETWORK 23
GVL.Led_Green_2 R= GVL.Seq_Done OR GVL.Man_Done;

// NETWORK 24
GVL.Led_Green_3 R= GVL.Seq_Done OR GVL.Man_Done;

// NETWORK 25
GVL.Led_Green_4 R= GVL.Seq_Done OR GVL.Man_Done;

// NETWORK 26
GVL.Led_Red_1 R= GVL.Seq_Done OR GVL.Man_Done;

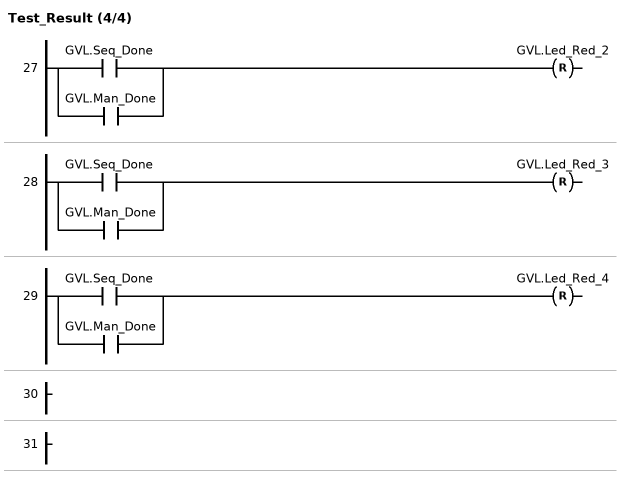
// NETWORK 27
GVL.Led_Red_2 R= GVL.Seq_Done OR GVL.Man_Done;

// NETWORK 28
GVL.Led_Red_3 R= GVL.Seq_Done OR GVL.Man_Done;

// NETWORK 29
GVL.Led_Red_4 R= GVL.Seq_Done OR GVL.Man_Done;

// NETWORK 30

// NETWORK 31

END_PROGRAM
